FUNCTION_BLOCK HMI_COME_TO_ME
  (* Standard: 61499-2 *)
  (* Version 1.0, 2018-12-12, adeel14a *)
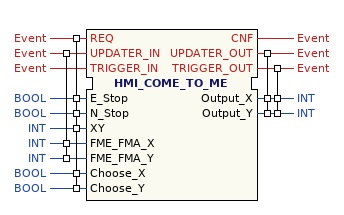
  EVENT_INPUT
    REQ WITH E_Stop, N_Stop, Choose_X, Choose_Y, XY;
    UPDATER_IN WITH FME_FMA_Y, FME_FMA_X;
    TRIGGER_IN;
  END_EVENT
  EVENT_OUTPUT
    CNF;
    UPDATER_OUT WITH Output_X, Output_Y;
    TRIGGER_OUT WITH Output_X, Output_Y;
  END_EVENT
  VAR_INPUT
    E_Stop : BOOL;
    N_Stop : BOOL;
    XY : INT;
    FME_FMA_X : INT;
    FME_FMA_Y : INT;
    Choose_X : BOOL;
    Choose_Y : BOOL;
  END_VAR
  VAR_OUTPUT
    Output_X : INT;
    Output_Y : INT;
  END_VAR
  SERVICE APPLICATION/RESOURCE
    SEQUENCE normal_establishment
      APPLICATION.INIT+(PARAMS) -> RESOURCE.initialize(PARAMS) -> APPLICATION.INITO+();
    END_SEQUENCE
    SEQUENCE unsuccessful_establishment
      APPLICATION.INIT+(PARAMS) -> RESOURCE.initialize(PARAMS) -> APPLICATION.INITO-(STATUS);
    END_SEQUENCE
    SEQUENCE request_confirm
      APPLICATION.REQ+(SD) -> RESOURCE.request(SD) -> APPLICATION.CNF+(RD);
    END_SEQUENCE
    SEQUENCE request_inhibited
      APPLICATION.REQ-(SD) -> APPLICATION.CNF-(STATUS);
    END_SEQUENCE
    SEQUENCE request_error
      APPLICATION.REQ+(SD) -> RESOURCE.request(SD) -> APPLICATION.CNF-(STATUS);
    END_SEQUENCE
    SEQUENCE indication_response
      RESOURCE.indicate(RD) -> APPLICATION.IND+(RD);
      APPLICATION.RSP(QI,SD) -> RESOURCE.response(QI,SD);
    END_SEQUENCE
    SEQUENCE indication_inhibited
      RESOURCE.indicate(RD,QI=FALSE) -> RESOURCE.inhibited();
    END_SEQUENCE
    SEQUENCE error_indication
      RESOURCE.error(STATUS) -> APPLICATION.IND-(STATUS);
    END_SEQUENCE
    SEQUENCE application_initiated_termination
      APPLICATION.INIT-() -> RESOURCE.terminate() -> APPLICATION.INITO-(STATUS);
    END_SEQUENCE
    SEQUENCE resource_initiated_termination
      -> APPLICATION.INITO-(STATUS);
    END_SEQUENCE
  END_SERVICE
END_FUNCTION_BLOCK
